Staubli VAL3: getSizeItem.pgx

public program getSizeItem(bool x_bCycle, num& x_nSize)
  local string l_sType
  local string l_sKey
  local num i
begin
  //
  // get the size of the collection
  //
  if x_bCycle
    x_nSize=size(pt:tTraj[sItemCycle].tData)
  else
    x_nSize=size(pEditPoint.tData)
  endIf
end
